// Brief: Master Arm Standby
FUNCTION_BLOCK PUBLIC FB_StateCtrlMountInstru EXTENDS FB_SlaveArmCtrlBase
VAR_INPUT
END_VAR
VAR_OUTPUT
END_VAR
VAR
	// mount status
	m_mountStatus :INT := 0;
	
	// flag if joint is mounted
	m_jointMounted :ARRAY[1..5] OF BOOL := [5(FALSE)];
	
	// instrument mount motion range
	m_mountMotionAng :Vec5d :=[1.25*PI, PI/2, PI/2, PI/2, PI/2];
	
	// instrument mount direction
	m_mountDir :Vec5i :=[1, 1, 1, 1, 1];
	
	// mount motion planning
	m_jntOTG :ARRAY[1..5] OF FB_secOrdTrajFilter;
	m_instruMountVel :LREAL := 30* g_deg2Rad;
	m_instruMountAcc :LREAL := PI;
	
	// track error threshold which indicate motor is buckled with panel
	m_maxTrackErr :LREAL := 5*g_deg2Rad;
	
	// command mount motion
	m_targetMountPos :Vec5d;
	
	// instrument zero position
	m_instruZeroPos :Vec5d;
END_VAR

// override this function in each exact controller
METHOD PROTECTED calcCmdJntPos : BOOL
VAR_INPUT
	motionScale :LREAL;
	masterIdx :INT;
END_VAR

VAR_IN_OUT CONSTANT
	i_slaveArm :FB_SlaveArm;
	i_masterStatus :ST_MasterStatus;
END_VAR

VAR 
	i :INT;
	curJntVel :Vec8d;
	curJntPos :Vec8d;
	jntPosErr :Vec8d;
END_VAR

curJntPos := i_slaveArm.curJntPos;

CASE m_mountStatus OF
	// To lock panel with instrument
	0:
		FOR i:=1 TO 5 DO
			// check joint buckled with instrument
			IF ABS(m_cmdJntPos[i+3]-curJntPos[i+3])> m_maxTrackErr THEN 
				m_jointMounted[i]:=TRUE;
				m_targetMountPos[i]:=curJntPos[i+3];
			END_IF
			
			// set target joint position
			IF FALSE = m_jointMounted[i] THEN
				// check mount motion direction
				IF ABS(m_cmdJntPos[i+3]-m_targetMountPos[i])< GVL_SlaveControlParameters.g_jntCtrlPosTol THEN
					m_mountDir[i]:=-1*m_mountDir[i];
				END_IF
				m_targetMountPos[i]:=m_mountDir[i]*m_mountMotionAng[i];
			END_IF
		END_FOR
		
		IF (m_jointMounted[1] AND m_jointMounted[2] AND m_jointMounted[3] AND m_jointMounted[4] AND m_jointMounted[5]) THEN
			m_mountStatus:=1;
		END_IF
	
	// determine zero position
	1:
		m_targetMountPos:=g_instruZeroPosition;
		m_mountStatus :=2;
	
	// move back to zero position
	2:
		vecSub(m_targetMountPos,curJntPos,jntPosErr);
		IF vecNorm(jntPosErr)<GVL_SlaveControlParameters.g_jntCtrlPosTol THEN
			m_isFinished:=TRUE;
		END_IF
END_CASE

// traj plan
FOR i:=1 TO 5 DO
	m_jntOTG[i].run(m_targetMountPos[i],0.0, o_cmdAcc=>m_cmdJntAcc[3+i],o_cmdVel=>m_cmdJntVel[3+i],o_cmdPos=>m_cmdJntPos[i+3]);
END_FOR
END_METHOD

METHOD PUBLIC init : BOOL
VAR_IN_OUT CONSTANT
	i_slaveArm	:FB_SlaveArm;
END_VAR
VAR_IN_OUT 
	r_slaveArmCtrlCmd :ST_SlaveArmCtrlCmds;
END_VAR
SUPER^.Init(i_slaveArm,r_slaveArmCtrlCmd);

// check if to hold the command joint position unchanged
checkToHoldLastCmds(i_slaveArm,r_slaveArmCtrlCmd);

// check instrument type to get mount joint index and zero position
IF i_slaveArm.instrument.instruType <> InstruType_UNKNOWM THEN
	m_jointMounted[5]:=TRUE;
	m_instruZeroPos[1]:=0;// need to update based on instrument type
	m_instruZeroPos[2]:=0;
	m_instruZeroPos[3]:=0;
	m_instruZeroPos[4]:=0;
	m_instruZeroPos[5]:=0;
END_IF
END_METHOD

END_FUNCTION_BLOCK

(* stored: Version 1.1.0.1, ProductVersion 3.1.4024.12
   POU FB_StateCtrlMountInstru: Id {db93de24-03af-45f5-8edb-e02a943fe1f8}, SpecialFunc None
   Method calcCmdJntPos: Id {106b8ce6-26fa-4bca-bfc9-20f8cdf00f0e}
   Method init: Id {85ccbdcb-d27d-4162-a6ec-e8e93d30dbc6} *)
